(* PLC project  *)

CONFIGURATION CiA402_Process_Data_1st
END_CONFIGURATION
